// TwinCAT 3 PLC project target_plc_proj
// ProgramVersion: 3.1.4023.0
// libraries:
//   L2SI Vacuum Library, * (SLAC)
//   LCLS General, * (SLAC)
//   Tc2_Standard, * (Beckhoff Automation GmbH)
//   Tc2_System, * (Beckhoff Automation GmbH)
//   Tc3_Module, * (Beckhoff Automation GmbH)
// project tree:
//   / PlcTask.TcTTO
//   POUs/ MAIN.TcPOU
// real-time tasks:
//   TASK PlcTask: cycle T#10ms, priority 20, ADS port 350
// I/O:
//   DEVICE Device 1 (EtherCAT), AmsNetId 5.54.18.118.2.1
//     Term 1 (EK1200) [EK1200-5000 EtherCAT Power supply (2A E-Bus)]
//       Term 2 (EL2212) [EL2212 2Ch. dig. output with overexcitation (24V DC, 2.5A, 10A Peak)]
//       Term 3 (EL1004) [EL1004 4Ch. Dig. Input 24V, 3ms]
//       Term 4 (EK1110) [EK1110 EtherCAT extension]

CONFIGURATION target_plc_proj
    RESOURCE PLC ON TwinCAT3
        TASK PlcTask(INTERVAL := T#10ms, PRIORITY := 20);
        PROGRAM MAIN WITH PlcTask : MAIN;
    END_RESOURCE
END_CONFIGURATION

// ---- POUs/MAIN.TcPOU
PROGRAM MAIN
VAR
	counter_x : INT := 0;
	
	test_gcc : FB_MKS422;
	test_vgc : FB_VGC;
	
	ads_watch_dog : FB_ADS_WATCHDOG;
END_VAR

// A counter to confirm that the program is running
IF counter_x < 1000 THEN
	counter_x := counter_x + 1;
ELSE
	counter_x := 0;
END_IF

//test_gcc();
//test_vgc();

(*
ads_watch_dog(
	sNetId:="5.54.18.118.1.1",
	nPort:=851,
	sVarName:="",
	bError:=
)
*)

END_PROGRAM
